Yaskawa INFORM job: HOME-POSITION-ROBOT-1.JBI

/JOB
//NAME HOME-POSITION-ROBOT-1
//POS
///NPOS 1,1,0,0,0,0
///TOOL 0
///POSTYPE PULSE
///PULSE
C00000=0,0,0,0,0,46844
BC00000=175235
//INST
///DATE 2018/09/06 14:03
///ATTR SC,RW
///GROUP1 RB1,BS1
NOP
MOVJ C00000 BC00000 VJ=10.00
TIMER T=1.00
END
